RoboDK station: New Station (2).rdk

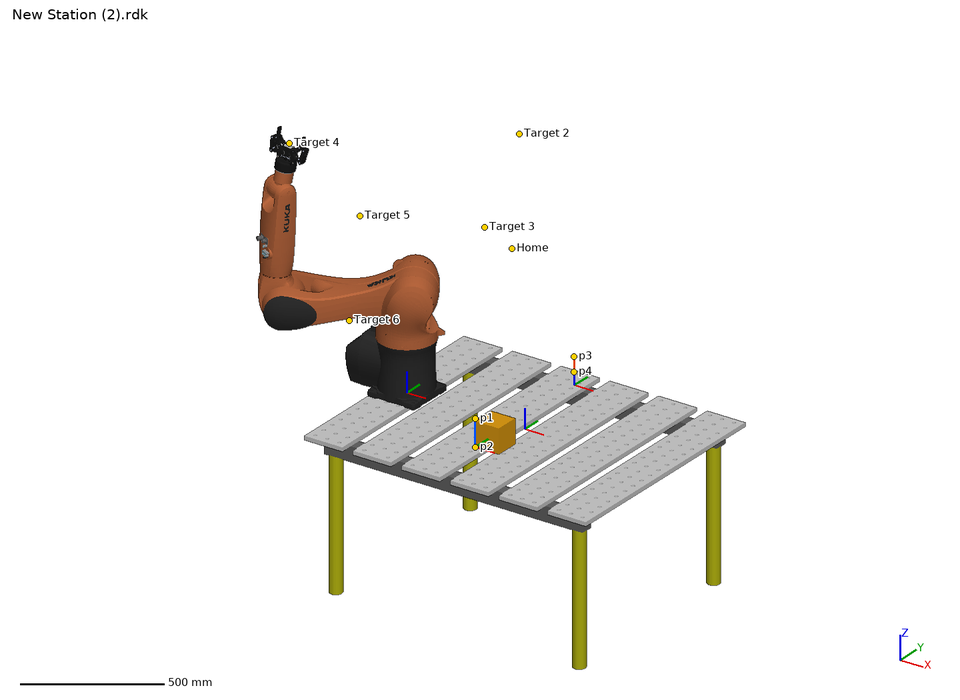
[picture v0: the station drawn from its stored meshes, robots at their saved joint values, targets as dots, program paths as lines]
Station New Station (2) (saved by RoboDK 5.9.0). Poses are relative to the parent item; angles as X-Y-Z fixed-axis rotations.
  - frame KUKA KR 10 R900 sixx Base at (-500, 0, 0) mm
    - robot KUKA KR 10 R900 sixx: 6 axes, payload 10 kg, reach 901 mm, repeatability 0.03 mm, weight 52 kg
        modified DH rows (alpha deg, a mm, theta deg, d mm): 0, 0, 0, 400; -90, 25, 0, 0; 0, 455, -90, 0; -90, 35, 0, 420; 90, 0, 0, 0; -90, 0, 180, 80
        joint limits [-170, -190, -120, -185, -120, -350] to [170, 45, 156, 185, 120, 350]; home [0, -90, 90, 0, 0, 0]; saved at [-32.123, -186.196, 99.512, -28.877, 7.409, -118.106]
      - tool RobotiQ 2F-85 Gripper (Open), TCP at (0, 0, 99.25) mm, size 147.4 x 75 x 146.8 mm
  - frame base at (0, 0, 0) mm
    - object Table 1200x1000mm (Welding) at (0, 0, 0) mm, size 1193.8 x 965.2 x 609.6 mm, geometry from Table-1200x1000mm-Welding.sld
    - target Home (Cartesian target) at (-55, 0, 680) mm, rotated rx 180 ry 0 rz -180 deg; joints [0, -90, 90, 0, 90, 0] of KUKA KR 10 R900 sixx
    - target Target 2 (Cartesian target) at (-325.76, 432.75, 876.68) mm, rotated rx -179.58 ry -6.24 rz 175.16 deg; joints [-23.682, -79.632, 54.934, -6.457, 117.018, -73.499] of KUKA KR 10 R900 sixx
    - target Target 3 (Cartesian target) at (-382.02, 301.85, 552.17) mm, rotated rx -177.39 ry -6.2 rz 171.06 deg; joints [-23.555, -101.897, 122.501, -5.498, 73.638, -72.791] of KUKA KR 10 R900 sixx
    - target Target 4 (Cartesian target) at (-851.05, -207.23, 948.5) mm, rotated rx 8.37 ry -6.26 rz 178.75 deg; joints [10.058, -186.196, 99.512, -28.877, 7.409, -118.106] of KUKA KR 10 R900 sixx
    - target Target 5 (Cartesian target) at (-397.93, -427.65, 882.97) mm, rotated rx -179.58 ry -6.24 rz 175.16 deg; joints [116.321, -83.164, 58.138, 6.703, 116.687, 72.248] of KUKA KR 10 R900 sixx
    - target Target 6 (Cartesian target) at (-443.7, -426.86, 465.38) mm, rotated rx -179.58 ry -6.24 rz 175.16 deg; joints [122.116, -84.562, 119.116, 7.337, 56.865, 71.026] of KUKA KR 10 R900 sixx
  - frame part1 at (0, -300, 50) mm
    - target p1 (Cartesian target) at (0, 0, 110) mm, rotated rx 180 ry 0 rz -180 deg; joints [30.964, -44.703, 105.627, 0, 29.076, 30.964] of KUKA KR 10 R900 sixx
    - target p2 (Cartesian target) at (0, 0, 0) mm, rotated rx 180 ry 0 rz -180 deg; joints [30.964, -32.411, 102.794, 0, 19.616, 30.964] of KUKA KR 10 R900 sixx
    - object Cube 100mm at (0, 0, 0) mm, size 100 x 100 x 100 mm, geometry from Cube-100mm.sld
  - frame part2 at (0, 300, 50) mm
    - target p3 (Cartesian target) at (0, 0, 110) mm, rotated rx 180 ry 0 rz -180 deg; joints [-30.964, -44.703, 105.627, 0, 29.076, -30.964] of KUKA KR 10 R900 sixx
    - target p4 (Cartesian target) at (0, 0, 50) mm, rotated rx 180 ry 0 rz -180 deg; joints [-30.964, -38.123, 104.533, 0, 23.59, -30.964] of KUKA KR 10 R900 sixx
  - program Prog1 (1 instructions, listed below)
  - program picking (6 instructions, listed below)
  - program place (6 instructions, listed below)
  - program main (7 instructions, listed below)
  - Python program Prog5 (listed below)
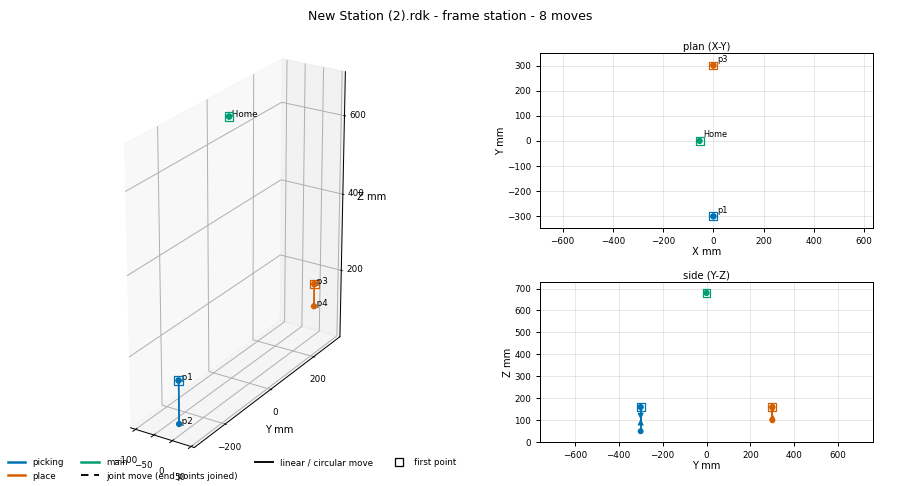
[picture p0: tool path of New Station (2).rdk in frame station, 8 of 8 moves have a stored position in this frame; points joined in program order, loops and branches not executed]

--- program Prog1 (robot KUKA KR 10 R900 sixx) ---
  Replace objects

--- program picking (robot KUKA KR 10 R900 sixx) ---
  Set Ref.: part1
  Set Tool: RobotiQ 2F-85 Gripper (Open)
  MoveJ (p1)
  MoveL (p2)
  Attach to RobotiQ 2F-85 Gripper (Open)
  MoveL (p1)

--- program place (robot KUKA KR 10 R900 sixx) ---
  Set Ref.: part2
  Set Tool: RobotiQ 2F-85 Gripper (Open)
  MoveJ (p3)
  MoveL (p4)
  Detach from RobotiQ 2F-85 Gripper (Open)
  MoveL (p3)

--- program main (robot KUKA KR 10 R900 sixx) ---
  Set Ref.: base
  Set Tool: RobotiQ 2F-85 Gripper (Open)
  MoveJ (Home)
  Call picking
  Call place
  Set Ref.: base
  MoveJ (Home)

--- Python program Prog5 ---
# Type help("robodk.robolink") or help("robodk.robomath") for more information
# Press F5 to run the script
# Documentation: https://robodk.com/doc/en/RoboDK-API.html
# Reference:     https://robodk.com/doc/en/PythonAPI/robodk.html
# Note: It is not required to keep a copy of this file, your Python script is saved with your RDK project

# You can also use the new version of the API:
from robodk import robolink    # RoboDK API
from robodk import robomath    # Robot toolbox
RDK = robolink.Robolink()

# Forward and backwards compatible use of the RoboDK API:
# Remove these 2 lines to follow python programming guidelines
from robodk import *      # RoboDK API
from robolink import *    # Robot toolbox
# Link to RoboDK
# RDK = Robolink()

# Notify user:
print('To edit this program:\nright click on the Python program, then, select "Edit Python script"')

# Program example:
item = RDK.Item('base')
if item.Valid():
    print('Item selected: ' + item.Name())
    print('Item posistion: ' + repr(item.Pose()))

print('Items in the station:')
itemlist = RDK.ItemList()
print(itemlist)

# Provoking an exception will display the console output if you run this script from RoboDK
raise Exception('Program not edited.')
